// TIA Portal V17 export
// export: Created 2025-06-26T06:49:30.1708255Z, ExportSetting WithDefaults, DisplayName Totally Integrated Automation Portal, DisplayVersion V17 Update 8, DisplayName TIA Portal Openness, DisplayVersion V17 Update 8, DisplayName TIA Portal Version Control Interface, DisplayVersion V17, DisplayName STEP 7 Professional, DisplayVersion V17 Update 8, DisplayName STEP 7 Safety, DisplayVersion V17 Update 6, DisplayName WinCC Advanced, DisplayVersion V17 Update 8
TYPE "stOnOffRegulator"
// stored: IsFailsafeCompliant false
   STRUCT
      bEnable : Bool;   // 1 = controller enabled, 0 = disabled
      fSetpoint : Real;   // Controller setpoint
      fHysteresis : Real := 0.5;   // Deadband around setpoint
      bOutput : Bool;   // 1 = output active
      bAtSetpoint : Bool;   // 1 = at setpoint
      bManualMode : Bool;   // 1 = activate manual mode
      fManualSetpoint : Real;   // Manual controller setpoint
      bManualOverride : Bool;   // 1 = activate override
      bOverrideCmd : Bool;   // 1 = force output on
      bFault : Bool;   // 1 = controller fault, 0 = ok
      nMode : USInt;   // 0 = Off, 1 = Auto, 2 = Manual, 3 = Manual Override
   END_STRUCT;
END_TYPE
